PROGRAM MAIN
VAR
    RandomDintValue		: LREAL;
	fbDRAND				: DRAND;
	
	start				: BOOL;
	timer1				: TON;
END_VAR

timer1(IN := start, PT := T#1S,);

start := TRUE;
IF timer1.Q THEN
	fbDRAND(Seed := 1);
	
	RandomDintValue := 100*fbDRAND.Num;
	start := FALSE;
END_IF;

END_PROGRAM

(* stored: Version 1.1.0.1, ProductVersion 3.1.4024.11
   POU MAIN: Id {72e0237f-1da5-48a1-99eb-6b55bdc0e73e}, SpecialFunc None *)
